(* PLC project Ladder.project, CODESYS CODESYS V3.5 SP15 *)
(* stored: creationDateTime 2020-02-10T18:54:44.558769, modificationDateTime 2020-02-10T18:28:58.901885 *)

PROGRAM PLC_PRG
VAR
	Variable: Int;
	NameEIGH: BOOL;
	Instance: FB_Name8;
END_VAR
  VAR  (* added by the conversion: wires and edge detectors of the diagram *)
    _F_Name5_Out01 : ANY;
    _F_Name5_Out02 : ANY;
    _F_Name5_OUT : BOOL;
    _w47 : BOOL;
  END_VAR

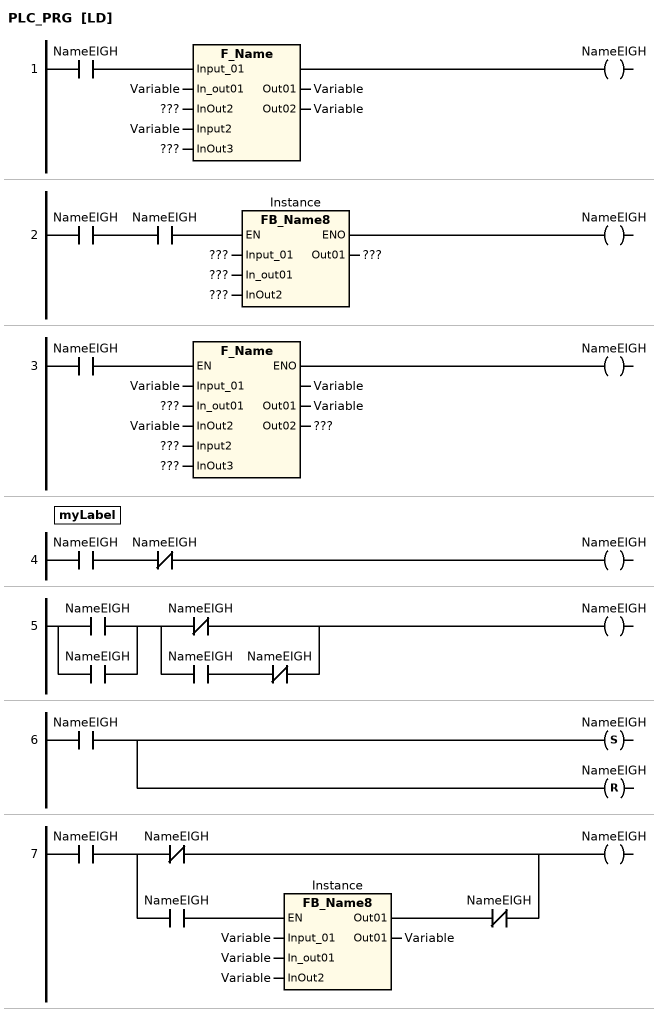
(* LD diagram, written out as Structured Text *)


_F_Name5_OUT := F_Name(Input_01 := NameEIGH, In_out01 := Variable, InOut2 := ???, Input2 := Variable, InOut3 := ???, Out01 => _F_Name5_Out01, Out02 => _F_Name5_Out02);
Variable := _F_Name5_Out01;
Variable := _F_Name5_Out02;
NameEIGH := _F_Name5_OUT;

Instance(EN := NameEIGH AND NameEIGH, Input_01 := ???, In_out01 := ???, InOut2 := ???, Out01 => ???);
NameEIGH := Instance.ENO;

IF NameEIGH THEN F_Name(Input_01 := Variable, In_out01 := ???, InOut2 := Variable, Input2 := ???, InOut3 := ???,     => Variable, Out01 => Variable, Out02 => ???); END_IF;
NameEIGH := NameEIGH;
myLabel:

NameEIGH := NameEIGH AND NOT NameEIGH;

NameEIGH := NameEIGH AND (NOT NameEIGH OR NameEIGH AND NOT NameEIGH);

_w47 := NameEIGH;
IF _w47 THEN NameEIGH := TRUE; END_IF;
IF _w47 THEN NameEIGH := FALSE; END_IF;

Instance(EN := NameEIGH AND NameEIGH, Input_01 := Variable, In_out01 := Variable, InOut2 := Variable, Out01 => Variable);
NameEIGH := NameEIGH AND NOT NameEIGH OR Instance.Out01 AND NOT NameEIGH;
(* --- network --- *)
END_PROGRAM
